{attribute 'qualified_only'}
{attribute 'strict'}
{attribute 'to_string'}
TYPE TRAFFIC_LIGHT_COLOR :
(
	NO_COLOR := 0,
	RED,
	YELLOW,
	GREEN
);
END_TYPE

(* stored: Version 1.1.0.1
   DUT TRAFFIC_LIGHT_COLOR: Id {ab9fe3a5-8110-4367-bf54-c77ad5d66b3a} *)
